FUNCTION_BLOCK FB_AnalogInputScaling_1
VAR_INPUT
	nRawInput 				: INT;
	stAnalogInputScaling    : ST_AnalogInputScaling;
END_VAR
VAR_OUTPUT
	fOutput 				: LREAL;
END_VAR
VAR
	fRawInput 				: LREAL;
	fNormalizedInput		: LREAL;
END_VAR

fRawInput := INT_TO_LREAL(nRawInput);

fNormalizedInput := (fRawInput - stAnalogInputScaling.fMinInputValue) / (stAnalogInputScaling.fMaxInputValue - stAnalogInputScaling.fMinInputValue);

fOutput := LIMIT(stAnalogInputScaling.fMinOutputValue, stAnalogInputScaling.fMinOutputValue + fNormalizedInput*(stAnalogInputScaling.fMaxOutputValue - stAnalogInputScaling.fMinOutputValue), stAnalogInputScaling.fMaxOutputValue);

END_FUNCTION_BLOCK

(* stored: Version 1.1.0.1, ProductVersion 3.1.4024.12
   POU FB_AnalogInputScaling_1: Id {cd5dbe47-ff67-4c1a-8ada-efe2e2de5501}, SpecialFunc None *)
